INTERFACE I_Contactor

METHOD Extend
VAR_INPUT
END_VAR
END_METHOD

PROPERTY Extended : BOOL
GET
END_GET
END_PROPERTY

PROPERTY ExtendTime : LREAL
GET
END_GET
SET
END_SET
END_PROPERTY

METHOD Retract
VAR_INPUT
END_VAR
END_METHOD

PROPERTY Retracted : BOOL
GET
END_GET
END_PROPERTY

PROPERTY RetractTime : LREAL
GET
END_GET
SET
END_SET
END_PROPERTY

END_INTERFACE

(* stored: Version 1.1.0.1, ProductVersion 3.1.4024.15
   Itf I_Contactor: Id {21f7d2a4-5739-4adf-9b0d-52a46ff8c7bf}
   Method Extend: Id {d98b7989-dd75-4631-8b18-2e1e4c76bd31}
   Property Extended: Id {727ecbc6-a446-451c-8abe-e65d679cf4da}
   Get Get: Id {ac822102-e49b-4fdf-9062-ec444370b38a}
   Property ExtendTime: Id {2c279e1d-c8d0-4217-a250-8a7a1f268f60}
   Get Get: Id {6ad4de30-7051-4ac6-8853-79b7416cb2b7}
   Set Set: Id {f7a7f276-1853-4d35-a9da-02a9e883b254}
   Method Retract: Id {4339714f-f15d-42e9-9aa6-fbd795c2634c}
   Property Retracted: Id {7ecd514d-3227-4478-b4cd-d9ab1bf67e1b}
   Get Get: Id {e9ba57b6-cd7b-4db9-99fd-e2e3dfef1393}
   Property RetractTime: Id {862a0ab4-5164-4785-8ea0-220c299c2b86}
   Get Get: Id {fe3c25d7-c590-4a6d-80f0-cf0361e6e874}
   Set Set: Id {b262f58e-c074-4e87-b2fe-3ab990c6c667} *)
